Fanuc KAREL source: kt00906.KL

PROGRAM KT00906
%STACKSIZE=65535
%PRIORITY=65535
%NOLOCKGROUP
VAR
P1 : JOINTPOS9
P2 : JOINTPOS9
OUT : VECTOR
BEGIN
-- UNSAFE_SOURCE_IR line 9: OUT = APPROACH(convert_jointpos9_to_position(P1))
END KT00906
